INTERFACE IMover EXTENDS __SYSTEM.IQueryInterface

PROPERTY AxisRef : reference to axis_ref
GET
END_GET
END_PROPERTY

METHOD DisableAxis : BOOL
VAR_INPUT
END_VAR
END_METHOD

METHOD EnableAxis : BOOL
VAR_INPUT
END_VAR
END_METHOD

METHOD HaltAxis : BOOL
VAR_INPUT
END_VAR
END_METHOD

METHOD HasCommand : BOOL
VAR_INPUT
END_VAR
END_METHOD

METHOD hasError : BOOL
VAR_INPUT
END_VAR
END_METHOD

PROPERTY IdentInGroup : int
GET
END_GET
SET
END_SET
END_PROPERTY

METHOD isAtPosition : BOOL
VAR_INPUT
	position : MC_LREAL;
END_VAR
END_METHOD

METHOD isDetected : BOOL
VAR_INPUT
END_VAR
END_METHOD

METHOD isEnabled : BOOL
VAR_INPUT
END_VAR
END_METHOD

METHOD isPastPosition : BOOL
VAR_INPUT
	position : MC_LREAL;
END_VAR
END_METHOD

METHOD isStationary : BOOL
VAR_INPUT
END_VAR
END_METHOD

METHOD MoveTo : BOOL
VAR_INPUT
	Position : MC_LREAL;
	Velocity : MC_LREAL;
	BackwardMove : BOOL;
END_VAR
END_METHOD

METHOD ResetAxis : BOOL
VAR_INPUT
END_VAR
END_METHOD

END_INTERFACE

(* stored: Version 1.1.0.1, ProductVersion 3.1.4024.12
   Itf IMover: Id {ee4a9524-17a3-415c-8258-028cd907ec8e}
   Property AxisRef: Id {f65c735e-9b12-45ca-8eb0-8081a48b017c}
   Get Get: Id {b5388ae2-ec1e-43b8-b87d-e490ff43d651}
   Method DisableAxis: Id {98eb94e3-2a36-4f82-9be2-aad46958ad3a}
   Method EnableAxis: Id {f0793d43-86f5-4db0-a1fc-77899ed18f09}
   Method HaltAxis: Id {6ff511eb-9b1d-4cc2-b90b-691594d634d8}
   Method HasCommand: Id {ec17e903-af29-44bd-a98a-e815b76d1aa3}
   Method hasError: Id {22eac0ed-a635-4f3d-8360-bc3525f3c471}
   Property IdentInGroup: Id {e90f3052-fcde-431f-9a44-66336e7806fd}
   Get Get: Id {75524577-6f6f-40a0-b905-f99e1140fc7f}
   Set Set: Id {d1d2db7b-41e7-42c7-be87-99aa9492a2ef}
   Method isAtPosition: Id {0a7edf6e-8fa0-440d-b312-6ae2eba5f40e}
   Method isDetected: Id {88edb286-cce8-49a5-b3bd-e1be274603b6}
   Method isEnabled: Id {9c1ac701-2fc5-4606-9f16-19eafb548c61}
   Method isPastPosition: Id {3b48a939-0d8a-43e9-aac7-eb23bcc49362}
   Method isStationary: Id {030c291b-8ff0-4518-9870-61eebdd699b2}
   Method MoveTo: Id {d70784c5-4dea-4741-b17d-2731466a43d5}
   Method ResetAxis: Id {86c2937f-07fa-4c6d-affc-f247383989e8} *)
